// TIA Portal V19 export
DATA_BLOCK "_IOL_VM_Values"   // DB500
TITLE = IOL is short for IO-Link
{ S7_Optimized_Access := 'TRUE' }
// stored: AutoNumber false, MemoryReserve 0
   VAR RETAIN
      V0930 : "_IOL_VmData";
      V0931 : "_IOL_VmData";
      V0552 : "_IOL_VmData";
      V0934 : "_IOL_VmData";
      V0935 : "_IOL_VmData";
      V0940 : "_IOL_VmData";
      V0941 : "_IOL_VmData";
      V0942 : "_IOL_VmData";
      V0943 : "_IOL_VmData";
      V0944 : "_IOL_VmData";
      V0945 : "_IOL_VmData";
      V1021 : "_IOL_VmData";
      V1023 : "_IOL_VmData";
      V1024 : "_IOL_VmData";
      V1025 : "_IOL_VmData";
      V1027 : "_IOL_VmData";
      V1083 : "_IOL_VmData";
      V0936 : "_IOL_VmData";
   END_VAR
BEGIN
   V1024.ObjErrorTime := -7744;
END_DATA_BLOCK
